{attribute 'qualified_only' := ''}
{attribute 'strict' := ''}
TYPE cStatus :
(
	None := 0,
	Empty := 1,
	Full := 2,
	RejectMalformedAPIData := 98,
	Reject := 99
) DINT;
END_TYPE

(* stored: Version 1.1.0.1, ProductVersion 3.1.4024.6
   DUT cStatus: Id {9e49f9eb-fe91-456e-b110-0b32065695fa} *)
